PROGRAM Emergency_Stop
VAR
	Stop_Button:BOOL;
END_VAR

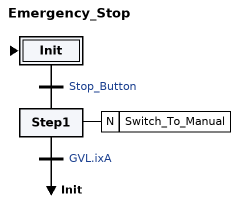
INITIAL_STEP Init:
END_STEP
TRANSITION FROM Init TO Step1
    := Stop_Button;
END_TRANSITION
STEP Step1:
    Switch_To_Manual(N);
END_STEP
TRANSITION FROM Step1 TO Init
    := GVL.ixA;
END_TRANSITION

ACTION Switch_To_Manual:
Automatic_Or_Manual.Automatic_Or_Manual:=FALSE;
END_ACTION

END_PROGRAM

(* stored: Version 1.1.0.1, ProductVersion 3.1.4024.12
   POU Emergency_Stop: Id {99e84d18-ee72-470a-b33b-22249ec199e8}, SpecialFunc None
   Action Switch_To_Manual: Id {5fd73dbf-9cdd-416f-a72e-073cf1f066b7} *)
